FUNCTION_BLOCK ASR_TO_ASR2 (* Composite FB for convert unidirectional ASR to bidirectional ASR2 *)
  (* Standard: 61499-2; Function: ASR_IN publishes SET/RESET onto the outgoing (EO_SET/EO_RESET) side of ASR2_BIDIR. Whatever ASR2_BIDIR receives on its incoming (EI_SET/EI_RESET) side is forwarded out again as plain unidirectional SET/RESET events via ASR_OUT.; Description: Copyright (c) 2026 HR Agrartechnik GmbH This program and the accompanying materials are made available under the terms of the Eclipse Public License 2.0 which is available at https://www.eclipse.org/legal/epl-2.0/ SPDX-License-Identifier: EPL-2.0 *)
  (* Version 1.0, 2026-08-31, Franz Höpfinger, HR Agrartechnik GmbH, Initial Version *)
  PACKAGE adapter::conversion::bidirectional;
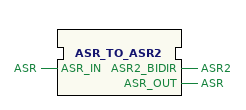
  SOCKETS
    ASR_IN : adapter::types::unidirectional::ASR; (* Adapter Input: unidirectional source *)
  END_SOCKETS
  PLUGS
    ASR2_BIDIR : adapter::types::bidirectional::ASR2; (* Adapter Output: bidirectional tap, outgoing side driven by ASR_IN, incoming side forwarded to ASR_OUT *)
    ASR_OUT : adapter::types::unidirectional::ASR; (* Adapter Output: mirrors ASR2_BIDIR's incoming (request) side *)
  END_PLUGS
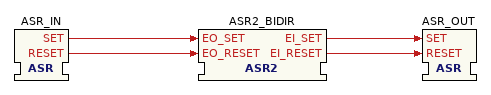
  EVENT_CONNECTIONS
    ASR_IN.SET TO ASR2_BIDIR.EO_SET;
    ASR_IN.RESET TO ASR2_BIDIR.EO_RESET;
    ASR2_BIDIR.EI_SET TO ASR_OUT.SET;
    ASR2_BIDIR.EI_RESET TO ASR_OUT.RESET;
  END_CONNECTIONS
END_FUNCTION_BLOCK
